{attribute addProperty BoxType "AT2050-5500-0018"}
{attribute addProperty Id "StatusAT %I*UINT1621Value_ChannelAT %I*ARRAY[0 ..31] OF INT512640"}
{attribute addProperty CRC "2166626233"}
{attribute addProperty SizeInBites "528"}
{attribute addProperty SizeInBytes "66"}
TYPE FB_Inputs_A6E87AE0 :
STRUCT
	{attribute addProperty Name "Status"}
	Status AT %I* : UINT;
	{attribute addProperty Name "Value_Channel"}
	Value_Channel AT %I* : ARRAY[0 ..31] OF INT;
END_STRUCT
END_TYPE

(* stored: Version 1.2.0.0, ProductVersion 3.1.4024.9
   DUT FB_Inputs_A6E87AE0: Id {7ddbf1b7-481d-450f-895f-cc3c98e701e2} *)
